Staubli VAL3: decodeLocation.pgx

program decodeLocation(point& value, num& buffer[])
  local num decodeBuffer[6]
begin
  fromBinary(buffer, 24, "4.0b", decodeBuffer)

  value.trsf = {decodeBuffer[0], decodeBuffer[1], decodeBuffer[2], decodeBuffer[3], decodeBuffer[4], decodeBuffer[5]}

  logMsg("P: (" + toString("3", value.trsf.x) + ", " + toString("3", value.trsf.y) + ", " + toString("3", value.trsf.z) + ")  R: (" + toString("3", value.trsf.rx) + ", " + toString("3", value.trsf.ry) + ", " + toString("3", value.trsf.rz) + ")")
end
